{attribute 'GeneratedUsingTerminal: KL3351'}
{attribute addProperty BoxType "KL3351"}
{attribute addProperty Id "StatusAT %I*USINT0Ud_RegInAT %I*INT0UrefAT %I*INT0CtrlAT %Q*USINT0RegOutAT %Q*INT0"}
{attribute addProperty CRC "765722428"}
{attribute addProperty Size "0"}
TYPE Channel_2DA3FF3C :
STRUCT
	{attribute addProperty Name "Status"}
	Status AT %I* : USINT;
	{attribute addProperty Name "Ud_RegIn"}
	Ud_RegIn AT %I* : INT;
	{attribute addProperty Name "Uref"}
	Uref AT %I* : INT;
	{attribute addProperty Name "Ctrl"}
	Ctrl AT %Q* : USINT;
	{attribute addProperty Name "RegOut"}
	RegOut AT %Q* : INT;
END_STRUCT
END_TYPE

(* stored: Version 1.2.0.0, ProductVersion 3.1.4024.9
   DUT Channel_2DA3FF3C: Id {13f7d3bd-077a-414c-abfd-243daa255f35} *)
